// TwinCAT 3 PLC project Quality_Analyzer
// ProgramVersion: 3.1.4024.0
// libraries:
//   Tc2_Standard, * (Beckhoff Automation GmbH)
//   Tc2_System, * (Beckhoff Automation GmbH)
//   Tc3_Module, * (Beckhoff Automation GmbH)
// project tree:
//   DUTs/ ST_ProductStats.TcDUT
//   / PlcTask.TcTTO
//   POUs/ AnalayzeBatch.TcPOU, CalculateAverage.TcPOU, CountDefects.TcPOU, FindMinMax.TcPOU, MAIN.TcPOU
// real-time tasks:
//   TASK PlcTask: cycle T#10ms, priority 20, ADS port 350

CONFIGURATION Quality_Analyzer
    RESOURCE PLC ON TwinCAT3
        TASK PlcTask(INTERVAL := T#10ms, PRIORITY := 20);
        PROGRAM MAIN WITH PlcTask : MAIN;
    END_RESOURCE
END_CONFIGURATION

// ---- DUTs/ST_ProductStats.TcDUT
TYPE ST_ProductStats :
STRUCT
	fAverageWeight : REAL;
	fminWeight : REAL;
	fmaxWeight : REAL;
	nDefectiveCount : INT;
END_STRUCT
END_TYPE

// ---- POUs/MAIN.TcPOU
PROGRAM MAIN
VAR
aProductArray : ARRAY[1..20] OF REAL := [23,120,35,100,250,300,500,230,190,30,10,600,240,210,10000,8600,11,349.444,42.252,534.2];
stProductAnalysis : ST_ProductStats;
END_VAR

stProductAnalysis := AnalayzeBatch(aProductArray);

END_PROGRAM

// ---- POUs/AnalayzeBatch.TcPOU
FUNCTION AnalayzeBatch : ST_ProductStats
VAR_INPUT
	aProdArray : REFERENCE TO ARRAY[1..20] OF REAL ;
END_VAR
VAR
	
END_VAR


AnalayzeBatch.fAverageWeight := CalculateAverage(aProdArray);
FindMinMax(aProdArray, nMinWeight => AnalayzeBatch.fminWeight, nMaxWeight => AnalayzeBatch.fmaxWeight);
AnalayzeBatch.nDefectiveCount := CountDefects(aProdArray);

END_FUNCTION

// ---- POUs/CalculateAverage.TcPOU
FUNCTION CalculateAverage : REAL
VAR_INPUT
END_VAR
VAR_IN_OUT
	aRefArray : ARRAY[1..20] OF REAL;
END_VAR
VAR
	nSum : REAL := 0;
	nIterator : INT;
END_VAR

FOR nIterator := 1 TO 20 DO
	nSum := nSum + aRefArray[nIterator];
END_FOR

CalculateAverage := nSum / 20;

END_FUNCTION

// ---- POUs/FindMinMax.TcPOU
FUNCTION FindMinMax : REAL
VAR_INPUT
END_VAR
VAR_IN_OUT
	aRefArray : ARRAY[1..20] OF REAL;
END_VAR
VAR
	nIterator : INT;
END_VAR
VAR_OUTPUT
	fMinWeight : REAL ;
	fMaxWeight : REAL;
END_VAR


fMinWeight := aRefArray[1];
fMaxWeight := aRefArray[1];
FOR nIterator := 2 TO 20 DO
	IF aRefArray[nIterator] < fMinWeight THEN
		fMinWeight := aRefArray[nIterator];
	END_IF
	IF aRefArray[nIterator] > fMaxWeight THEN
		fMaxWeight := aRefArray[nIterator];
	END_IF
END_FOR

END_FUNCTION

// ---- POUs/CountDefects.TcPOU
FUNCTION CountDefects : INT
VAR_INPUT
	aRefArray : REFERENCE TO ARRAY[1..20] OF REAL;
END_VAR
VAR
	
	nIterator: INT;
END_VAR

FOR nIterator := 1 TO 20 DO
	IF aRefArray[nIterator] < 50 THEN
		CountDefects := CountDefects + 1;
	END_IF
	IF aRefArray[nIterator] > 500 THEN
		CountDefects := CountDefects + 1;
	END_IF
END_FOR

END_FUNCTION
